{attribute 'qualified_only'}
{attribute 'to_string'}
TYPE E_GCSingleProcessStage :
(
	None := 0,
	Prepare := 1,
	LiftReady := 2,
	SpinAlign := 3,
	ConcurrentProcessEntry := 4,
	SpinRampUp := 5,
	ProcessHold := 6,
	ConcurrentProcessExit := 7,
	SpinStandby := 8
) UINT;
END_TYPE

(* stored: Version 1.1.0.1, ProductVersion 3.1.4026.18
   DUT E_GCSingleProcessStage: Id {7df990a2-494a-40ba-b4cb-804b3ee52003} *)
